ABB RobotStudio station: Project_Lab2.rspag

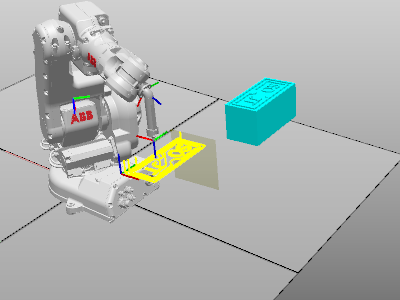
--- station ---
Station Project1 (saved by RobotStudio 25.1.11167.1)
Controller Controller_Lab2
  mechanical unit ROB_1: IRB140_6_81_C_03, 6 joints, base frame (0, 0, 0) mm
Layout (positions relative to the parent item):
  - IRB140_6_81_C_03 [mechanism, from %ABB.RobotStudio.Models.IRB140%\IRB140_6_81_C_G_03.rslib] at (0, 0, 0) mm; joint values [2.6873, 0.1595, -0.1337, 0.7807, 0.6006, -0.8887] (rad or m)
  - Marcador_2 [mechanism, from Project_Lab2\Marcador.rslib] at (-514.53, 222.5, 670.16) mm, rotated rx 180 ry 65 rz 0 deg
  - Pastel [part] at (-541.34, 72.5, 291.55) mm, rotated rx 5 ry 0 rz 90 deg, size 300 x 140 x 145 mm
  - SmartComponent_3 [smart component]
      signals: DI DI_SM01, DO DO_SM01, DI DI_SM03
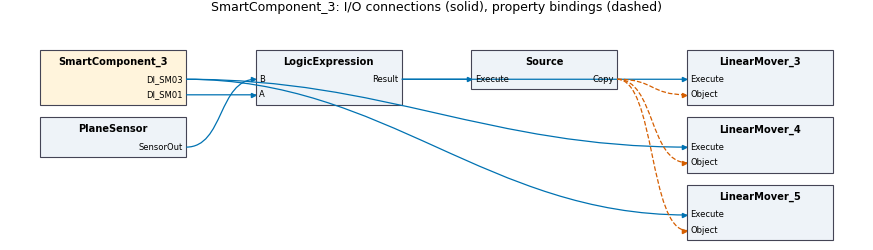
      connections:
        LogicExpression.Result -> Source.Execute
        LogicExpression.Result -> LinearMover_3.Execute
        SmartComponent_3.DI_SM03 -> LinearMover_4.Execute
        PlaneSensor.SensorOut -> LogicExpression.B
        SmartComponent_3.DI_SM01 -> LogicExpression.A
        SmartComponent_3.DI_SM03 -> LinearMover_5.Execute
        Source.Copy => LinearMover_4.Object
        Source.Copy => LinearMover_3.Object
        Source.Copy => LinearMover_5.Object
    - PlaneSensor [smart component, from Components\PlaneSensor.rslib] at (-518.61, 72.5, 264.47) mm, rotated rx 5 ry 0 rz 90 deg
        properties: Origin=[0 0 0]; Axis1=[0 0.19 0]; Axis2=[0 0 0.195]; Tag=(none); SenseMultiple=false; SensedPart=(none)
      - _sensorPart_ [part], size 0 x 190 x 195 mm
    - LinearMover_3 [smart component, from Components\LinearMover.rslib]
        properties: Object=Pastel_2; Direction=[0 -0.1 0]; Speed=0.05; Reference=Global; ReferenceObject=(none)
    - Source [smart component, from Components\Source.rslib]
        properties: Source=Pastel; Copy=Pastel_2; Parent=(none); Position=[-0.5413376 0.3225 0.2915518]; Orientation=[0.0872664625997165 0 1.5707963267949]; Transient=false; PhysicsBehavior=-1
    - LogicExpression [smart component, from Components\LogicExpression.rslib]
        properties: Expression=(A AND (NOT B))
    - LinearMover_5 [smart component, from Components\LinearMover.rslib]
        properties: Object=Pastel_2; Direction=[0 -0.1 0]; Speed=0.2; Reference=Global; ReferenceObject=(none)
  - Pastel_2 [part] at (-541.34, -532.5, 291.55) mm, rotated rx 5 ry 0 rz 90 deg, size 300 x 140 x 145 mm
Attachment: Marcador_2 is attached to IRB140_6_81_C_03 / Link6
Station logic (signal -> signal, property => property):
  Controller_Lab2.DO_01 -> SmartComponent_3.DI_SM01
  Controller_Lab2.vDO_03 -> SmartComponent_3.DI_SM03

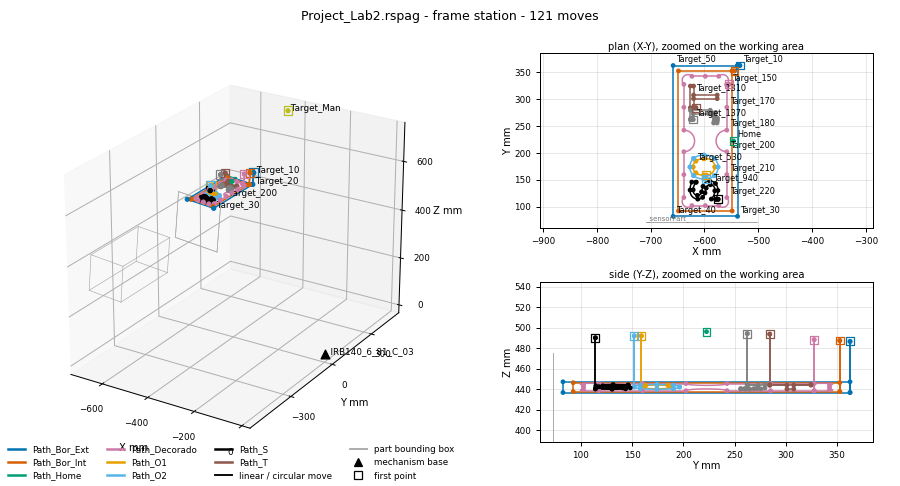
[picture p0: tool path of Project_Lab2.rspag in frame station, 121 of 121 moves have a stored position in this frame; points joined in program order, loops and branches not executed]
--- Controller Data/Controller_Lab2/RAPID/TASK1/PROGMOD/CalibData.mod ---
MODULE CalibData
ENDMODULE

--- Controller Data/Controller_Lab2/RAPID/TASK1/PROGMOD/Module1.mod ---
MODULE Module1
    PERS tooldata TCP_Marcador:=[TRUE,[[144.332,0,101.99],[0.866025404,0,0.5,0]],[1,[0,0,1],[1,0,0,0],0,0,0]];
    CONST robtarget Target_240:=[[45,270,0],[0.130526192,0,0.991444861,0],[0,0,0,0],[9E+09,9E+09,9E+09,9E+09,9E+09,9E+09]];
    CONST robtarget Target_10:=[[10,10,50],[0.130526192,0,0.991444861,0],[0,0,0,0],[9E+09,9E+09,9E+09,9E+09,9E+09,9E+09]];
    CONST robtarget Target_20:=[[10,10,0],[0.130526192,0,0.991444861,0],[0,0,0,0],[9E+09,9E+09,9E+09,9E+09,9E+09,9E+09]];
    CONST robtarget Target_30:=[[10,290,0],[0.130526192,0,0.991444861,0],[0,0,0,0],[9E+09,9E+09,9E+09,9E+09,9E+09,9E+09]];
    CONST robtarget Target_40:=[[130,290,0],[0.130526192,0,0.991444861,0],[0,0,0,0],[9E+09,9E+09,9E+09,9E+09,9E+09,9E+09]];
    CONST robtarget Target_50:=[[130,10,0],[0.130526192,0,0.991444861,0],[0,0,0,0],[9E+09,9E+09,9E+09,9E+09,9E+09,9E+09]];
    CONST robtarget Target_60:=[[10,10,0],[0.130526192,0,0.991444861,0],[0,0,0,0],[9E+09,9E+09,9E+09,9E+09,9E+09,9E+09]];
    CONST robtarget Target_70:=[[10,10,50],[0.130526192,0,0.991444861,0],[0,0,0,0],[9E+09,9E+09,9E+09,9E+09,9E+09,9E+09]];
    CONST robtarget Target_80:=[[20,20,50],[0.130526192,0,0.991444861,0],[0,0,0,0],[9E+09,9E+09,9E+09,9E+09,9E+09,9E+09]];
    CONST robtarget Target_90:=[[20,20,0],[0.130526192,0,0.991444861,0],[0,0,0,0],[9E+09,9E+09,9E+09,9E+09,9E+09,9E+09]];
    CONST robtarget Target_100:=[[20,280,0],[0.130526192,0,0.991444861,0],[0,0,0,0],[9E+09,9E+09,9E+09,9E+09,9E+09,9E+09]];
    CONST robtarget Target_110:=[[120,280,0],[0.130526192,0,0.991444861,0],[0,0,0,0],[9E+09,9E+09,9E+09,9E+09,9E+09,9E+09]];
    CONST robtarget Target_120:=[[120,20,0],[0.130526192,0,0.991444861,0],[0,0,0,0],[9E+09,9E+09,9E+09,9E+09,9E+09,9E+09]];
    CONST robtarget Target_130:=[[20,20,0],[0.130526192,0,0.991444861,0],[0,0,0,0],[9E+09,9E+09,9E+09,9E+09,9E+09,9E+09]];
    CONST robtarget Target_140:=[[20,20,50],[0.130526192,0,0.991444861,0],[0,0,0,0],[9E+09,9E+09,9E+09,9E+09,9E+09,9E+09]];
    CONST robtarget Target_150:=[[30,45,50],[0.130526192,0,0.991444861,0],[0,0,0,0],[9E+09,9E+09,9E+09,9E+09,9E+09,9E+09]];
    CONST robtarget Target_160:=[[30,45,0],[0.130526192,0,0.991444861,0],[0,0,0,0],[9E+09,9E+09,9E+09,9E+09,9E+09,9E+09]];
    CONST robtarget Target_170:=[[30,87.5,0],[0.130526192,0,0.991444861,0],[0,0,0,0],[9E+09,9E+09,9E+09,9E+09,9E+09,9E+09]];
    CONST robtarget Target_180:=[[30,130,0],[0.130526192,0,0.991444861,0],[0,0,0,0],[9E+09,9E+09,9E+09,9E+09,9E+09,9E+09]];
    CONST robtarget Target_190:=[[50,150,0],[0.130526192,0,0.991444861,0],[0,0,0,0],[9E+09,9E+09,9E+09,9E+09,9E+09,9E+09]];
    CONST robtarget Target_200:=[[30,170,0],[0.130526192,0,0.991444861,0],[0,0,0,0],[9E+09,9E+09,9E+09,9E+09,9E+09,9E+09]];
    CONST robtarget Target_210:=[[30,212.5,0],[0.130526192,0,0.991444861,0],[0,0,0,0],[9E+09,9E+09,9E+09,9E+09,9E+09,9E+09]];
    CONST robtarget Target_220:=[[30,255,0],[0.130526192,0,0.991444861,0],[0,0,0,0],[9E+09,9E+09,9E+09,9E+09,9E+09,9E+09]];
    CONST robtarget Target_230:=[[30,270,0],[0.130526192,0,0.991444861,0],[0,0,0,0],[9E+09,9E+09,9E+09,9E+09,9E+09,9E+09]];
    TASK PERS wobjdata Workobject_pastel:=[FALSE,TRUE,"",[[-528.7,372.5,436],[0,0.043619387,0,0.999048222]],[[0,0,0],[1,0,0,0]]];
    CONST robtarget Home:=[[22.451582178,150,58.509821421],[0,0,1,0],[0,0,0,0],[9E+09,9E+09,9E+09,9E+09,9E+09,9E+09]];
    CONST robtarget Target_250:=[[70,270,0],[0.130526192,0,0.991444861,0],[0,0,0,0],[9E+09,9E+09,9E+09,9E+09,9E+09,9E+09]];
    CONST robtarget Target_260:=[[95,270,0],[0.130526192,0,0.991444861,0],[0,0,0,0],[9E+09,9E+09,9E+09,9E+09,9E+09,9E+09]];
    CONST robtarget Target_270:=[[110,270,0],[0.130526192,0,0.991444861,0],[0,0,0,0],[9E+09,9E+09,9E+09,9E+09,9E+09,9E+09]];
    CONST robtarget Target_280:=[[110,255,0],[0.130526192,0,0.991444861,0],[0,0,0,0],[9E+09,9E+09,9E+09,9E+09,9E+09,9E+09]];
    CONST robtarget Target_290:=[[110,212.5,0],[0.130526192,0,0.991444861,0],[0,0,0,0],[9E+09,9E+09,9E+09,9E+09,9E+09,9E+09]];
    CONST robtarget Target_300:=[[110,170,0],[0.130526192,0,0.991444861,0],[0,0,0,0],[9E+09,9E+09,9E+09,9E+09,9E+09,9E+09]];
    CONST robtarget Target_310:=[[90,150,0],[0.130526192,0,0.991444861,0],[0,0,0,0],[9E+09,9E+09,9E+09,9E+09,9E+09,9E+09]];
    CONST robtarget Target_320:=[[110,130,0],[0.130526192,0,0.991444861,0],[0,0,0,0],[9E+09,9E+09,9E+09,9E+09,9E+09,9E+09]];
    CONST robtarget Target_330:=[[110,87.5,0],[0.130526192,0,0.991444861,0],[0,0,0,0],[9E+09,9E+09,9E+09,9E+09,9E+09,9E+09]];
    CONST robtarget Target_340:=[[110,45,0],[0.130526192,0,0.991444861,0],[0,0,0,0],[9E+09,9E+09,9E+09,9E+09,9E+09,9E+09]];
    CONST robtarget Target_350:=[[110,30,0],[0.130526192,0,0.991444861,0],[0,0,0,0],[9E+09,9E+09,9E+09,9E+09,9E+09,9E+09]];
    CONST robtarget Target_360:=[[95,30,0],[0.130526192,0,0.991444861,0],[0,0,0,0],[9E+09,9E+09,9E+09,9E+09,9E+09,9E+09]];
    CONST robtarget Target_370:=[[70,30,0],[0.130526192,0,0.991444861,0],[0,0,0,0],[9E+09,9E+09,9E+09,9E+09,9E+09,9E+09]];
    CONST robtarget Target_380:=[[45,30,0],[0.130526192,0,0.991444861,0],[0,0,0,0],[9E+09,9E+09,9E+09,9E+09,9E+09,9E+09]];
    CONST robtarget Target_390:=[[30,30,0],[0.130526192,0,0.991444861,0],[0,0,0,0],[9E+09,9E+09,9E+09,9E+09,9E+09,9E+09]];
    CONST robtarget Target_400:=[[30,45,0],[0.130526192,0,0.991444861,0],[0,0,0,0],[9E+09,9E+09,9E+09,9E+09,9E+09,9E+09]];
    CONST robtarget Target_410:=[[30,45,50],[0.130526192,0,0.991444861,0],[0,0,0,0],[9E+09,9E+09,9E+09,9E+09,9E+09,9E+09]];
    CONST robtarget Target_420:=[[72.5,213.529,50],[0.130526192,0,0.991444861,0],[0,0,0,0],[9E+09,9E+09,9E+09,9E+09,9E+09,9E+09]];
    CONST robtarget Target_430:=[[72.5,213.529,0],[0.130526192,0,0.991444861,0],[0,0,0,0],[9E+09,9E+09,9E+09,9E+09,9E+09,9E+09]];
    CONST robtarget Target_440:=[[57.427,209.396,0],[0.130526192,0,0.991444861,0],[0,0,0,0],[9E+09,9E+09,9E+09,9E+09,9E+09,9E+09]];
    CONST robtarget Target_450:=[[52.2,198.335,0],[0.130526192,0,0.991444861,0],[0,0,0,0],[9E+09,9E+09,9E+09,9E+09,9E+09,9E+09]];
    CONST robtarget Target_460:=[[52.2,198.335,0],[0.130526192,0,0.991444861,0],[0,0,0,0],[9E+09,9E+09,9E+09,9E+09,9E+09,9E+09]];
    CONST robtarget Target_470:=[[57.427,187.293,0],[0.130526192,0,0.991444861,0],[0,0,0,0],[9E+09,9E+09,9E+09,9E+09,9E+09,9E+09]];
    CONST robtarget Target_480:=[[72.5,183.181,0],[0.130526192,0,0.991444861,0],[0,0,0,0],[9E+09,9E+09,9E+09,9E+09,9E+09,9E+09]];
    CONST robtarget Target_490:=[[72.5,183.181,0],[0.130526192,0,0.991444861,0],[0,0,0,0],[9E+09,9E+09,9E+09,9E+09,9E+09,9E+09]];
    CONST robtarget Target_500:=[[81.272,184.254,0],[0.130526192,0,0.991444861,0],[0,0,0,0],[9E+09,9E+09,9E+09,9E+09,9E+09,9E+09]];
    CONST robtarget Target_510:=[[87.613,187.273,0],[0.130526192,0,0.991444861,0],[0,0,0,0],[9E+09,9E+09,9E+09,9E+09,9E+09,9E+09]];
    CONST robtarget Target_520:=[[87.613,187.273,0],[0.130526192,0,0.991444861,0],[0,0,0,0],[9E+09,9E+09,9E+09,9E+09,9E+09,9E+09]];
    CONST robtarget Target_530:=[[91.503,192.054,0],[0.130526192,0,0.991444861,0],[0,0,0,0],[9E+09,9E+09,9E+09,9E+09,9E+09,9E+09]];
    CONST robtarget Target_540:=[[92.8,198.335,0],[0.130526192,0,0.991444861,0],[0,0,0,0],[9E+09,9E+09,9E+09,9E+09,9E+09,9E+09]];
    CONST robtarget Target_550:=[[92.8,198.335,0],[0.130526192,0,0.991444861,0],[0,0,0,0],[9E+09,9E+09,9E+09,9E+09,9E+09,9E+09]];
    CONST robtarget Target_560:=[[91.544,204.656,0],[0.130526192,0,0.991444861,0],[0,0,0,0],[9E+09,9E+09,9E+09,9E+09,9E+09,9E+09]];
    CONST robtarget Target_570:=[[87.613,209.437,0],[0.130526192,0,0.991444861,0],[0,0,0,0],[9E+09,9E+09,9E+09,9E+09,9E+09,9E+09]];
    CONST robtarget Target_580:=[[87.613,209.437,0],[0.130526192,0,0.991444861,0],[0,0,0,0],[9E+09,9E+09,9E+09,9E+09,9E+09,9E+09]];
    CONST robtarget Target_590:=[[81.212,212.476,0],[0.130526192,0,0.991444861,0],[0,0,0,0],[9E+09,9E+09,9E+09,9E+09,9E+09,9E+09]];
    CONST robtarget Target_600:=[[72.5,213.529,0],[0.130526192,0,0.991444861,0],[0,0,0,0],[9E+09,9E+09,9E+09,9E+09,9E+09,9E+09]];
    CONST robtarget Target_610:=[[72.5,213.529,50],[0.130526192,0,0.991444861,0],[0,0,0,0],[9E+09,9E+09,9E+09,9E+09,9E+09,9E+09]];
    CONST robtarget Target_620:=[[72.5,220.458,50],[0.130526192,0,0.991444861,0],[0,0,0,0],[9E+09,9E+09,9E+09,9E+09,9E+09,9E+09]];
    CONST robtarget Target_630:=[[72.5,220.458,0],[0.130526192,0,0.991444861,0],[0,0,0,0],[9E+09,9E+09,9E+09,9E+09,9E+09,9E+09]];
    CONST robtarget Target_640:=[[61.459,218.918,0],[0.130526192,0,0.991444861,0],[0,0,0,0],[9E+09,9E+09,9E+09,9E+09,9E+09,9E+09]];
    CONST robtarget Target_650:=[[53.254,214.502,0],[0.130526192,0,0.991444861,0],[0,0,0,0],[9E+09,9E+09,9E+09,9E+09,9E+09,9E+09]];
    CONST robtarget Target_660:=[[53.254,214.502,0],[0.130526192,0,0.991444861,0],[0,0,0,0],[9E+09,9E+09,9E+09,9E+09,9E+09,9E+09]];
    CONST robtarget Target_670:=[[48.169,207.492,0],[0.130526192,0,0.991444861,0],[0,0,0,0],[9E+09,9E+09,9E+09,9E+09,9E+09,9E+09]];
    CONST robtarget Target_680:=[[46.447,198.375,0],[0.130526192,0,0.991444861,0],[0,0,0,0],[9E+09,9E+09,9E+09,9E+09,9E+09,9E+09]];
    CONST robtarget Target_690:=[[46.447,198.375,0],[0.130526192,0,0.991444861,0],[0,0,0,0],[9E+09,9E+09,9E+09,9E+09,9E+09,9E+09]];
    CONST robtarget Target_700:=[[48.108,189.4,0],[0.130526192,0,0.991444861,0],[0,0,0,0],[9E+09,9E+09,9E+09,9E+09,9E+09,9E+09]];
    CONST robtarget Target_710:=[[53.254,182.249,0],[0.130526192,0,0.991444861,0],[0,0,0,0],[9E+09,9E+09,9E+09,9E+09,9E+09,9E+09]];
    CONST robtarget Target_720:=[[53.254,182.249,0],[0.130526192,0,0.991444861,0],[0,0,0,0],[9E+09,9E+09,9E+09,9E+09,9E+09,9E+09]];
    CONST robtarget Target_730:=[[61.499,177.792,0],[0.130526192,0,0.991444861,0],[0,0,0,0],[9E+09,9E+09,9E+09,9E+09,9E+09,9E+09]];
    CONST robtarget Target_740:=[[72.5,176.252,0],[0.130526192,0,0.991444861,0],[0,0,0,0],[9E+09,9E+09,9E+09,9E+09,9E+09,9E+09]];
    CONST robtarget Target_750:=[[72.5,176.252,0],[0.130526192,0,0.991444861,0],[0,0,0,0],[9E+09,9E+09,9E+09,9E+09,9E+09,9E+09]];
    CONST robtarget Target_760:=[[83.602,177.832,0],[0.130526192,0,0.991444861,0],[0,0,0,0],[9E+09,9E+09,9E+09,9E+09,9E+09,9E+09]];
    CONST robtarget Target_770:=[[91.787,182.249,0],[0.130526192,0,0.991444861,0],[0,0,0,0],[9E+09,9E+09,9E+09,9E+09,9E+09,9E+09]];
    CONST robtarget Target_780:=[[91.787,182.249,0],[0.130526192,0,0.991444861,0],[0,0,0,0],[9E+09,9E+09,9E+09,9E+09,9E+09,9E+09]];
    CONST robtarget Target_790:=[[96.771,189.177,0],[0.130526192,0,0.991444861,0],[0,0,0,0],[9E+09,9E+09,9E+09,9E+09,9E+09,9E+09]];
    CONST robtarget Target_800:=[[98.553,198.375,0],[0.130526192,0,0.991444861,0],[0,0,0,0],[9E+09,9E+09,9E+09,9E+09,9E+09,9E+09]];
    CONST robtarget Target_810:=[[98.553,198.375,0],[0.130526192,0,0.991444861,0],[0,0,0,0],[9E+09,9E+09,9E+09,9E+09,9E+09,9E+09]];
    CONST robtarget Target_820:=[[96.831,207.472,0],[0.130526192,0,0.991444861,0],[0,0,0,0],[9E+09,9E+09,9E+09,9E+09,9E+09,9E+09]];
    CONST robtarget Target_830:=[[91.787,214.461,0],[0.130526192,0,0.991444861,0],[0,0,0,0],[9E+09,9E+09,9E+09,9E+09,9E+09,9E+09]];
    CONST robtarget Target_840:=[[91.787,214.461,0],[0.130526192,0,0.991444861,0],[0,0,0,0],[9E+09,9E+09,9E+09,9E+09,9E+09,9E+09]];
    CONST robtarget Target_850:=[[83.562,218.898,0],[0.130526192,0,0.991444861,0],[0,0,0,0],[9E+09,9E+09,9E+09,9E+09,9E+09,9E+09]];
    CONST robtarget Target_860:=[[72.5,220.458,0],[0.130526192,0,0.991444861,0],[0,0,0,0],[9E+09,9E+09,9E+09,9E+09,9E+09,9E+09]];
    CONST robtarget Target_870:=[[72.5,220.458,50],[0.130526192,0,0.991444861,0],[0,0,0,0],[9E+09,9E+09,9E+09,9E+09,9E+09,9E+09]];
    CONST robtarget Target_880:=[[50.498,258.383,50],[0.130526192,0,0.991444861,0],[0,0,0,0],[9E+09,9E+09,9E+09,9E+09,9E+09,9E+09]];
    CONST robtarget Target_890:=[[50.498,258.383,0],[0.130526192,0,0.991444861,0],[0,0,0,0],[9E+09,9E+09,9E+09,9E+09,9E+09,9E+09]];
    CONST robtarget Target_900:=[[58.845,257.897,0],[0.130526192,0,0.991444861,0],[0,0,0,0],[9E+09,9E+09,9E+09,9E+09,9E+09,9E+09]];
    CONST robtarget Target_910:=[[54.064,250.462,0],[0.130526192,0,0.991444861,0],[0,0,0,0],[9E+09,9E+09,9E+09,9E+09,9E+09,9E+09]];
    CONST robtarget Target_920:=[[52.362,242.459,0],[0.130526192,0,0.991444861,0],[0,0,0,0],[9E+09,9E+09,9E+09,9E+09,9E+09,9E+09]];
    CONST robtarget Target_930:=[[54.652,234.133,0],[0.130526192,0,0.991444861,0],[0,0,0,0],[9E+09,9E+09,9E+09,9E+09,9E+09,9E+09]];
    CONST robtarget Target_940:=[[60.709,231.317,0],[0.130526192,0,0.991444861,0],[0,0,0,0],[9E+09,9E+09,9E+09,9E+09,9E+09,9E+09]];
    CONST robtarget Target_950:=[[65.571,232.796,0],[0.130526192,0,0.991444861,0],[0,0,0,0],[9E+09,9E+09,9E+09,9E+09,9E+09,9E+09]];
    CONST robtarget Target_960:=[[68.367,237.476,0],[0.130526192,0,0.991444861,0],[0,0,0,0],[9E+09,9E+09,9E+09,9E+09,9E+09,9E+09]];
    CONST robtarget Target_970:=[[69.461,241.71,0],[0.130526192,0,0.991444861,0],[0,0,0,0],[9E+09,9E+09,9E+09,9E+09,9E+09,9E+09]];
    CONST robtarget Target_980:=[[70.636,246.511,0],[0.130526192,0,0.991444861,0],[0,0,0,0],[9E+09,9E+09,9E+09,9E+09,9E+09,9E+09]];
    CONST robtarget Target_990:=[[72.358,251.151,0],[0.130526192,0,0.991444861,0],[0,0,0,0],[9E+09,9E+09,9E+09,9E+09,9E+09,9E+09]];
    CONST robtarget Target_1000:=[[75.053,254.777,0],[0.130526192,0,0.991444861,0],[0,0,0,0],[9E+09,9E+09,9E+09,9E+09,9E+09,9E+09]];
    CONST robtarget Target_1010:=[[78.942,257.168,0],[0.130526192,0,0.991444861,0],[0,0,0,0],[9E+09,9E+09,9E+09,9E+09,9E+09,9E+09]];
    CONST robtarget Target_1020:=[[84.088,258.019,0],[0.130526192,0,0.991444861,0],[0,0,0,0],[9E+09,9E+09,9E+09,9E+09,9E+09,9E+09]];
    CONST robtarget Target_1030:=[[94.279,253.278,0],[0.130526192,0,0.991444861,0],[0,0,0,0],[9E+09,9E+09,9E+09,9E+09,9E+09,9E+09]];
    CONST robtarget Target_1040:=[[98.391,241.203,0],[0.130526192,0,0.991444861,0],[0,0,0,0],[9E+09,9E+09,9E+09,9E+09,9E+09,9E+09]];
    CONST robtarget Target_1050:=[[97.561,233.262,0],[0.130526192,0,0.991444861,0],[0,0,0,0],[9E+09,9E+09,9E+09,9E+09,9E+09,9E+09]];
    CONST robtarget Target_1060:=[[95.15,226.333,0],[0.130526192,0,0.991444861,0],[0,0,0,0],[9E+09,9E+09,9E+09,9E+09,9E+09,9E+09]];
    CONST robtarget Target_1070:=[[87.208,226.333,0],[0.130526192,0,0.991444861,0],[0,0,0,0],[9E+09,9E+09,9E+09,9E+09,9E+09,9E+09]];
    CONST robtarget Target_1080:=[[87.208,226.819,0],[0.130526192,0,0.991444861,0],[0,0,0,0],[9E+09,9E+09,9E+09,9E+09,9E+09,9E+09]];
    CONST robtarget Target_1090:=[[91.017,232.938,0],[0.130526192,0,0.991444861,0],[0,0,0,0],[9E+09,9E+09,9E+09,9E+09,9E+09,9E+09]];
    CONST robtarget Target_1100:=[[92.638,240.758,0],[0.130526192,0,0.991444861,0],[0,0,0,0],[9E+09,9E+09,9E+09,9E+09,9E+09,9E+09]];
    CONST robtarget Target_1110:=[[90.47,248.233,0],[0.130526192,0,0.991444861,0],[0,0,0,0],[9E+09,9E+09,9E+09,9E+09,9E+09,9E+09]];
    CONST robtarget Target_1120:=[[84.777,251.09,0],[0.130526192,0,0.991444861,0],[0,0,0,0],[9E+09,9E+09,9E+09,9E+09,9E+09,9E+09]];
    CONST robtarget Target_1130:=[[79.733,249.408,0],[0.130526192,0,0.991444861,0],[0,0,0,0],[9E+09,9E+09,9E+09,9E+09,9E+09,9E+09]];
    CONST robtarget Target_1140:=[[76.998,244.566,0],[0.130526192,0,0.991444861,0],[0,0,0,0],[9E+09,9E+09,9E+09,9E+09,9E+09,9E+09]];
    CONST robtarget Target_1150:=[[75.701,239.4,0],[0.130526192,0,0.991444861,0],[0,0,0,0],[9E+09,9E+09,9E+09,9E+09,9E+09,9E+09]];
    CONST robtarget Target_1160:=[[74.364,234.315,0],[0.130526192,0,0.991444861,0],[0,0,0,0],[9E+09,9E+09,9E+09,9E+09,9E+09,9E+09]];
    CONST robtarget Target_1170:=[[69.603,226.779,0],[0.130526192,0,0.991444861,0],[0,0,0,0],[9E+09,9E+09,9E+09,9E+09,9E+09,9E+09]];
    CONST robtarget Target_1180:=[[61.763,224.388,0],[0.130526192,0,0.991444861,0],[0,0,0,0],[9E+09,9E+09,9E+09,9E+09,9E+09,9E+09]];
    CONST robtarget Target_1190:=[[55.968,225.583,0],[0.130526192,0,0.991444861,0],[0,0,0,0],[9E+09,9E+09,9E+09,9E+09,9E+09,9E+09]];
    CONST robtarget Target_1200:=[[51.147,228.926,0],[0.130526192,0,0.991444861,0],[0,0,0,0],[9E+09,9E+09,9E+09,9E+09,9E+09,9E+09]];
    CONST robtarget Target_1210:=[[47.784,234.356,0],[0.130526192,0,0.991444861,0],[0,0,0,0],[9E+09,9E+09,9E+09,9E+09,9E+09,9E+09]];
    CONST robtarget Target_1220:=[[46.609,241.973,0],[0.130526192,0,0.991444861,0],[0,0,0,0],[9E+09,9E+09,9E+09,9E+09,9E+09,9E+09]];
    CONST robtarget Target_1230:=[[47.743,251.212,0],[0.130526192,0,0.991444861,0],[0,0,0,0],[9E+09,9E+09,9E+09,9E+09,9E+09,9E+09]];
    CONST robtarget Target_1240:=[[50.498,258.383,0],[0.130526192,0,0.991444861,0],[0,0,0,0],[9E+09,9E+09,9E+09,9E+09,9E+09,9E+09]];
    CONST robtarget Target_1250:=[[50.498,258.383,50],[0.130526192,0,0.991444861,0],[0,0,0,0],[9E+09,9E+09,9E+09,9E+09,9E+09,9E+09]];
    CONST robtarget Target_1260:=[[91.929,88.314,50],[0.130526192,0,0.991444861,0],[0,0,0,0],[9E+09,9E+09,9E+09,9E+09,9E+09,9E+09]];
    CONST robtarget Target_1270:=[[91.929,88.314,0],[0.130526192,0,0.991444861,0],[0,0,0,0],[9E+09,9E+09,9E+09,9E+09,9E+09,9E+09]];
    CONST robtarget Target_1280:=[[97.844,88.314,0],[0.130526192,0,0.991444861,0],[0,0,0,0],[9E+09,9E+09,9E+09,9E+09,9E+09,9E+09]];
    CONST robtarget Target_1290:=[[97.844,48.12,0],[0.130526192,0,0.991444861,0],[0,0,0,0],[9E+09,9E+09,9E+09,9E+09,9E+09,9E+09]];
    CONST robtarget Target_1300:=[[91.929,48.12,0],[0.130526192,0,0.991444861,0],[0,0,0,0],[9E+09,9E+09,9E+09,9E+09,9E+09,9E+09]];
    CONST robtarget Target_1310:=[[91.929,64.895,0],[0.130526192,0,0.991444861,0],[0,0,0,0],[9E+09,9E+09,9E+09,9E+09,9E+09,9E+09]];
    CONST robtarget Target_1320:=[[47.844,64.895,0],[0.130526192,0,0.991444861,0],[0,0,0,0],[9E+09,9E+09,9E+09,9E+09,9E+09,9E+09]];
    CONST robtarget Target_1330:=[[47.844,71.54,0],[0.130526192,0,0.991444861,0],[0,0,0,0],[9E+09,9E+09,9E+09,9E+09,9E+09,9E+09]];
    CONST robtarget Target_1340:=[[91.929,71.54,0],[0.130526192,0,0.991444861,0],[0,0,0,0],[9E+09,9E+09,9E+09,9E+09,9E+09,9E+09]];
    CONST robtarget Target_1350:=[[91.929,88.314,0],[0.130526192,0,0.991444861,0],[0,0,0,0],[9E+09,9E+09,9E+09,9E+09,9E+09,9E+09]];
    CONST robtarget Target_1360:=[[91.929,88.314,50],[0.130526192,0,0.991444861,0],[0,0,0,0],[9E+09,9E+09,9E+09,9E+09,9E+09,9E+09]];
    CONST robtarget Target_1370:=[[97.844,110.235,50],[0.130526192,0,0.991444861,0],[0,0,0,0],[9E+09,9E+09,9E+09,9E+09,9E+09,9E+09]];
    CONST robtarget Target_1380:=[[97.844,110.235,0],[0.130526192,0,0.991444861,0],[0,0,0,0],[9E+09,9E+09,9E+09,9E+09,9E+09,9E+09]];
    CONST robtarget Target_1390:=[[97.844,93.015,0],[0.130526192,0,0.991444861,0],[0,0,0,0],[9E+09,9E+09,9E+09,9E+09,9E+09,9E+09]];
    CONST robtarget Target_1400:=[[60.851,93.015,0],[0.130526192,0,0.991444861,0],[0,0,0,0],[9E+09,9E+09,9E+09,9E+09,9E+09,9E+09]];
    CONST robtarget Target_1410:=[[50.721,97.026,0],[0.130526192,0,0.991444861,0],[0,0,0,0],[9E+09,9E+09,9E+09,9E+09,9E+09,9E+09]];
    CONST robtarget Target_1420:=[[47.156,107.804,0],[0.130526192,0,0.991444861,0],[0,0,0,0],[9E+09,9E+09,9E+09,9E+09,9E+09,9E+09]];
    CONST robtarget Target_1430:=[[47.439,112.119,0],[0.130526192,0,0.991444861,0],[0,0,0,0],[9E+09,9E+09,9E+09,9E+09,9E+09,9E+09]];
    CONST robtarget Target_1440:=[[48.128,116.637,0],[0.130526192,0,0.991444861,0],[0,0,0,0],[9E+09,9E+09,9E+09,9E+09,9E+09,9E+09]];
    CONST robtarget Target_1450:=[[54.53,116.637,0],[0.130526192,0,0.991444861,0],[0,0,0,0],[9E+09,9E+09,9E+09,9E+09,9E+09,9E+09]];
    CONST robtarget Target_1460:=[[53.476,112.848,0],[0.130526192,0,0.991444861,0],[0,0,0,0],[9E+09,9E+09,9E+09,9E+09,9E+09,9E+09]];
    CONST robtarget Target_1470:=[[52.909,108.695,0],[0.130526192,0,0.991444861,0],[0,0,0,0],[9E+09,9E+09,9E+09,9E+09,9E+09,9E+09]];
    CONST robtarget Target_1480:=[[53.618,103.772,0],[0.130526192,0,0.991444861,0],[0,0,0,0],[9E+09,9E+09,9E+09,9E+09,9E+09,9E+09]];
    CONST robtarget Target_1490:=[[55.624,101.078,0],[0.130526192,0,0.991444861,0],[0,0,0,0],[9E+09,9E+09,9E+09,9E+09,9E+09,9E+09]];
    CONST robtarget Target_1500:=[[58.906,99.903,0],[0.130526192,0,0.991444861,0],[0,0,0,0],[9E+09,9E+09,9E+09,9E+09,9E+09,9E+09]];
    CONST robtarget Target_1510:=[[63.404,99.66,0],[0.130526192,0,0.991444861,0],[0,0,0,0],[9E+09,9E+09,9E+09,9E+09,9E+09,9E+09]];
    CONST robtarget Target_1520:=[[92.536,99.66,0],[0.130526192,0,0.991444861,0],[0,0,0,0],[9E+09,9E+09,9E+09,9E+09,9E+09,9E+09]];
    CONST robtarget Target_1530:=[[92.536,110.235,0],[0.130526192,0,0.991444861,0],[0,0,0,0],[9E+09,9E+09,9E+09,9E+09,9E+09,9E+09]];
    CONST robtarget Target_1540:=[[97.844,110.235,0],[0.130526192,0,0.991444861,0],[0,0,0,0],[9E+09,9E+09,9E+09,9E+09,9E+09,9E+09]];
    CONST robtarget Target_1550:=[[97.844,110.235,50],[0.130526192,0,0.991444861,0],[0,0,0,0],[9E+09,9E+09,9E+09,9E+09,9E+09,9E+09]];
    CONST robtarget Target_Mantenimiento:=[[-1037.356401001,150,-97.894390869],[0,0.923879532,0,-0.382683432],[-2,0,0,1],[9E+09,9E+09,9E+09,9E+09,9E+09,9E+09]];
    CONST robtarget Target_Man:=[[-54.840948466,-101.359051534,293.521625448],[0.562422225,0.303603179,0.732962913,-0.232962913],[1,0,-1,1],[9E+09,9E+09,9E+09,9E+09,9E+09,9E+09]];



    PROC main()
        Reset DO_01;
        Reset DO_02;
        !Reset vDO_03;
        WHILE TRUE DO
            IF DI_01 = 1 THEN
                ! Arranque
                Set DO_01;      ! Variador de frecuencia y Linear Mover 1
                WaitTime 5;
                ! Freno
                Reset DO_01;

                ! Dibujar
                dibujar;

                ! Arranque
                Set DO_01;
                WaitTime 5;
                ! Freno
                Reset DO_01;

                ! Arranque
                Set vDO_03;     ! Smart Component
                WaitTime 3;
                ! Freno
                Reset vDO_03;
            ELSEIF DI_02 = 1 THEN
                Reset DO_01;
                Set DO_02;
                Path_Mantenimiento;
                WaitTime 1;
                Reset DO_02;
            ENDIF
        ENDWHILE
    ENDPROC

    PROC dibujar()
        Path_Home;
        WaitTime 2;
        Path_Bor_Ext;
        WaitTime 2;
        Path_Bor_Int;
        WaitTime 2;
        Path_Decorado;
        WaitTime 2;
        Path_S;
        WaitTime 2;
        Path_O1;
        WaitTime 2;
        Path_O2;
        WaitTime 2;
        Path_J;
        WaitTime 2;
        Path_T;
        WaitTime 2;
        Path_Home;
    ENDPROC

    PROC Path_Bor_Ext()
        MoveJ Target_10,v100,z10,TCP_Marcador\WObj:=Workobject_pastel;
        MoveL Target_20,v100,z10,TCP_Marcador\WObj:=Workobject_pastel;
        MoveL Target_30,v100,z10,TCP_Marcador\WObj:=Workobject_pastel;
        MoveL Target_40,v100,z10,TCP_Marcador\WObj:=Workobject_pastel;
        MoveL Target_50,v100,z10,TCP_Marcador\WObj:=Workobject_pastel;
        MoveL Target_60,v100,z10,TCP_Marcador\WObj:=Workobject_pastel;
        MoveL Target_70,v100,z10,TCP_Marcador\WObj:=Workobject_pastel;
    ENDPROC

    PROC Path_Bor_Int()
        MoveJ Target_80,v100,z10,TCP_Marcador\WObj:=Workobject_pastel;
        MoveL Target_90,v100,z10,TCP_Marcador\WObj:=Workobject_pastel;
        MoveL Target_100,v100,z10,TCP_Marcador\WObj:=Workobject_pastel;
        MoveL Target_110,v100,z10,TCP_Marcador\WObj:=Workobject_pastel;
        MoveL Target_120,v100,z10,TCP_Marcador\WObj:=Workobject_pastel;
        MoveL Target_130,v100,z10,TCP_Marcador\WObj:=Workobject_pastel;
        MoveL Target_140,v100,z10,TCP_Marcador\WObj:=Workobject_pastel;
    ENDPROC

    PROC Path_Home()
        MoveJ Home,v100,z10,TCP_Marcador\WObj:=Workobject_pastel;
    ENDPROC

    PROC Path_Decorado()
        MoveJ Target_150,v100,z10,TCP_Marcador\WObj:=Workobject_pastel;
        MoveL Target_160,v100,z10,TCP_Marcador\WObj:=Workobject_pastel;
        MoveL Target_170,v100,z10,TCP_Marcador\WObj:=Workobject_pastel;
        MoveL Target_180,v100,z10,TCP_Marcador\WObj:=Workobject_pastel;
        MoveC Target_190,Target_200,v100,z10,TCP_Marcador\WObj:=Workobject_pastel;
        MoveL Target_210,v100,z10,TCP_Marcador\WObj:=Workobject_pastel;
        MoveL Target_220,v100,z10,TCP_Marcador\WObj:=Workobject_pastel;
        MoveC Target_230,Target_240,v100,z10,TCP_Marcador\WObj:=Workobject_pastel;
        MoveL Target_250,v100,z10,TCP_Marcador\WObj:=Workobject_pastel;
        MoveL Target_260,v100,z10,TCP_Marcador\WObj:=Workobject_pastel;
        MoveC Target_270,Target_280,v100,z10,TCP_Marcador\WObj:=Workobject_pastel;
        MoveL Target_290,v100,z10,TCP_Marcador\WObj:=Workobject_pastel;
        MoveL Target_300,v100,z10,TCP_Marcador\WObj:=Workobject_pastel;
        MoveC Target_310,Target_320,v100,z10,TCP_Marcador\WObj:=Workobject_pastel;
        MoveL Target_330,v100,z10,TCP_Marcador\WObj:=Workobject_pastel;
        MoveL Target_340,v100,z10,TCP_Marcador\WObj:=Workobject_pastel;
        MoveC Target_350,Target_360,v100,z10,TCP_Marcador\WObj:=Workobject_pastel;
        MoveL Target_370,v100,z10,TCP_Marcador\WObj:=Workobject_pastel;
        MoveL Target_380,v100,z10,TCP_Marcador\WObj:=Workobject_pastel;
        MoveC Target_390,Target_400,v100,z10,TCP_Marcador\WObj:=Workobject_pastel;
        MoveL Target_410,v100,z10,TCP_Marcador\WObj:=Workobject_pastel;
    ENDPROC

    PROC Path_O1()
        MoveJ Target_420,v100,z10,TCP_Marcador\WObj:=Workobject_pastel;
        MoveL Target_430,v100,z10,TCP_Marcador\WObj:=Workobject_pastel;
        MoveC Target_440,Target_450,v100,z10,TCP_Marcador\WObj:=Workobject_pastel;
        MoveL Target_460,v100,z10,TCP_Marcador\WObj:=Workobject_pastel;
        MoveC Target_470,Target_480,v100,z10,TCP_Marcador\WObj:=Workobject_pastel;
        MoveL Target_490,v100,z10,TCP_Marcador\WObj:=Workobject_pastel;
        MoveC Target_500,Target_510,v100,z10,TCP_Marcador\WObj:=Workobject_pastel;
        MoveL Target_520,v100,z10,TCP_Marcador\WObj:=Workobject_pastel;
        MoveC Target_530,Target_540,v100,z10,TCP_Marcador\WObj:=Workobject_pastel;
        MoveL Target_550,v100,z10,TCP_Marcador\WObj:=Workobject_pastel;
        MoveC Target_560,Target_570,v100,z10,TCP_Marcador\WObj:=Workobject_pastel;
        MoveL Target_580,v100,z10,TCP_Marcador\WObj:=Workobject_pastel;
        MoveC Target_590,Target_600,v100,z10,TCP_Marcador\WObj:=Workobject_pastel;
        MoveL Target_610,v100,z10,TCP_Marcador\WObj:=Workobject_pastel;
    ENDPROC

    PROC Path_O2()
        MoveJ Target_620,v100,z10,TCP_Marcador\WObj:=Workobject_pastel;
        MoveL Target_630,v100,z10,TCP_Marcador\WObj:=Workobject_pastel;
        MoveC Target_640,Target_650,v100,z10,TCP_Marcador\WObj:=Workobject_pastel;
        MoveL Target_660,v100,z10,TCP_Marcador\WObj:=Workobject_pastel;
        MoveC Target_670,Target_680,v100,z10,TCP_Marcador\WObj:=Workobject_pastel;
        MoveL Target_690,v100,z10,TCP_Marcador\WObj:=Workobject_pastel;
        MoveC Target_700,Target_710,v100,z10,TCP_Marcador\WObj:=Workobject_pastel;
        MoveL Target_720,v100,z10,TCP_Marcador\WObj:=Workobject_pastel;
        MoveC Target_730,Target_740,v100,z10,TCP_Marcador\WObj:=Workobject_pastel;
        MoveL Target_750,v100,z10,TCP_Marcador\WObj:=Workobject_pastel;
        MoveC Target_760,Target_770,v100,z10,TCP_Marcador\WObj:=Workobject_pastel;
        MoveL Target_780,v100,z10,TCP_Marcador\WObj:=Workobject_pastel;
        MoveC Target_790,Target_800,v100,z10,TCP_Marcador\WObj:=Workobject_pastel;
        MoveL Target_810,v100,z10,TCP_Marcador\WObj:=Workobject_pastel;
        MoveC Target_820,Target_830,v100,z10,TCP_Marcador\WObj:=Workobject_pastel;
        MoveL Target_840,v100,z10,TCP_Marcador\WObj:=Workobject_pastel;
        MoveC Target_850,Target_860,v100,z10,TCP_Marcador\WObj:=Workobject_pastel;
        MoveL Target_870,v100,z10,TCP_Marcador\WObj:=Workobject_pastel;
    ENDPROC

    PROC Path_S()
        MoveJ Target_880,v100,z10,TCP_Marcador\WObj:=Workobject_pastel;
        MoveL Target_890,v100,z10,TCP_Marcador\WObj:=Workobject_pastel;
        MoveL Target_900,v100,z10,TCP_Marcador\WObj:=Workobject_pastel;
        MoveC Target_910,Target_920,v100,z10,TCP_Marcador\WObj:=Workobject_pastel;
        MoveC Target_930,Target_940,v100,z10,TCP_Marcador\WObj:=Workobject_pastel;
        MoveC Target_950,Target_960,v100,z10,TCP_Marcador\WObj:=Workobject_pastel;
        MoveC Target_970,Target_980,v100,z10,TCP_Marcador\WObj:=Workobject_pastel;
        MoveC Target_990,Target_1000,v100,z10,TCP_Marcador\WObj:=Workobject_pastel;
        MoveC Target_1010,Target_1020,v100,z10,TCP_Marcador\WObj:=Workobject_pastel;
        MoveC Target_1030,Target_1040,v100,z10,TCP_Marcador\WObj:=Workobject_pastel;
        MoveC Target_1050,Target_1060,v100,z10,TCP_Marcador\WObj:=Workobject_pastel;
        MoveL Target_1070,v100,z10,TCP_Marcador\WObj:=Workobject_pastel;
        MoveL Target_1080,v100,z10,TCP_Marcador\WObj:=Workobject_pastel;
        MoveC Target_1090,Target_1100,v100,z10,TCP_Marcador\WObj:=Workobject_pastel;
        MoveC Target_1110,Target_1120,v100,z10,TCP_Marcador\WObj:=Workobject_pastel;
        MoveC Target_1130,Target_1140,v100,z10,TCP_Marcador\WObj:=Workobject_pastel;
        MoveC Target_1150,Target_1160,v100,z10,TCP_Marcador\WObj:=Workobject_pastel;
        MoveC Target_1170,Target_1180,v100,z10,TCP_Marcador\WObj:=Workobject_pastel;
        MoveC Target_1190,Target_1200,v100,z10,TCP_Marcador\WObj:=Workobject_pastel;
        MoveC Target_1210,Target_1220,v100,z10,TCP_Marcador\WObj:=Workobject_pastel;
        MoveC Target_1230,Target_1240,v100,z10,TCP_Marcador\WObj:=Workobject_pastel;
        MoveL Target_1250,v100,z10,TCP_Marcador\WObj:=Workobject_pastel;
    ENDPROC

    PROC Path_T()
        MoveJ Target_1260,v100,z10,TCP_Marcador\WObj:=Workobject_pastel;
        MoveL Target_1270,v100,z10,TCP_Marcador\WObj:=Workobject_pastel;
        MoveL Target_1280,v100,z10,TCP_Marcador\WObj:=Workobject_pastel;
        MoveL Target_1290,v100,z10,TCP_Marcador\WObj:=Workobject_pastel;
        MoveL Target_1300,v100,z10,TCP_Marcador\WObj:=Workobject_pastel;
        MoveL Target_1310,v100,z10,TCP_Marcador\WObj:=Workobject_pastel;
        MoveL Target_1320,v100,z10,TCP_Marcador\WObj:=Workobject_pastel;
        MoveL Target_1330,v100,z10,TCP_Marcador\WObj:=Workobject_pastel;
        MoveL Target_1340,v100,z10,TCP_Marcador\WObj:=Workobject_pastel;
        MoveL Target_1350,v100,z10,TCP_Marcador\WObj:=Workobject_pastel;
        MoveL Target_1360,v100,z10,TCP_Marcador\WObj:=Workobject_pastel;
    ENDPROC

    PROC Path_J()
        MoveL Target_1370,v100,z10,TCP_Marcador\WObj:=Workobject_pastel;
        MoveL Target_1380,v100,z10,TCP_Marcador\WObj:=Workobject_pastel;
        MoveL Target_1390,v100,z10,TCP_Marcador\WObj:=Workobject_pastel;
        MoveL Target_1400,v100,z10,TCP_Marcador\WObj:=Workobject_pastel;
        MoveL Target_1410,v100,z10,TCP_Marcador\WObj:=Workobject_pastel;
        MoveL Target_1420,v100,z10,TCP_Marcador\WObj:=Workobject_pastel;
        MoveL Target_1430,v100,z10,TCP_Marcador\WObj:=Workobject_pastel;
        MoveL Target_1440,v100,z10,TCP_Marcador\WObj:=Workobject_pastel;
        MoveL Target_1450,v100,z10,TCP_Marcador\WObj:=Workobject_pastel;
        MoveL Target_1460,v100,z10,TCP_Marcador\WObj:=Workobject_pastel;
        MoveL Target_1470,v100,z10,TCP_Marcador\WObj:=Workobject_pastel;
        MoveL Target_1480,v100,z10,TCP_Marcador\WObj:=Workobject_pastel;
        MoveL Target_1490,v100,z10,TCP_Marcador\WObj:=Workobject_pastel;
        MoveL Target_1500,v100,z10,TCP_Marcador\WObj:=Workobject_pastel;
        MoveL Target_1510,v100,z10,TCP_Marcador\WObj:=Workobject_pastel;
        MoveL Target_1520,v100,z10,TCP_Marcador\WObj:=Workobject_pastel;
        MoveL Target_1530,v100,z10,TCP_Marcador\WObj:=Workobject_pastel;
        MoveL Target_1540,v100,z10,TCP_Marcador\WObj:=Workobject_pastel;
        MoveL Target_1550,v100,z10,TCP_Marcador\WObj:=Workobject_pastel;
    ENDPROC
    PROC Path_Mantenimiento()
        MoveJ Target_Man,v100,z10,TCP_Marcador\WObj:=Workobject_pastel;
    ENDPROC

ENDMODULE

--- Controller Data/Controller_Lab2/SYSPAR/EIO.cfg ---
EIO:CFG_1.0:6:1::
#
EIO_SIGNAL:

      -Name "DI_01" -SignalType "DI"

      -Name "DI_02" -SignalType "DI"

      -Name "DO_01" -SignalType "DO"

      -Name "DO_02" -SignalType "DO"

      -Name "vDO_03" -SignalType "DO"
